Fanuc KAREL source: ka00119.KL

-- PROVISIONAL review KL for V1013-1; original PC SHA256 0b4e37eaa532840a0307d8d150ba9d81eed41656d6312ba72b29ab2837e931de
-- Incomplete behavior may be omitted. Consult companion uncertainty JSON. Do not deploy.
PROGRAM KA00119
%NOLOCKGROUP
-- UNRESOLVED_DECL SRC type=00001c
-- UNRESOLVED_DECL DST type=002018
BEGIN
  -- UNRESOLVED_PC offsets 5-15; opcodes 9D,22,A5
  -- UNRESOLVED_PC offsets 20-35; opcodes 21,22,9D,33,B2
  -- UNRESOLVED_PC offsets 40-44; opcodes 7F
END KA00119
